(* LS Electric XG5000 project: 찐찐찐찐최종본_스마트홈_프로젝트_0225 *)
(* PLC LSPLC *)

(* Comments on direct variables
%MX0	램프0
%MX1	램프1
%MX2	램프2
%MX3	램프3
%MX4	색상조절변경버튼
%MX9	전원
%MX10	온도_자동
%MX11	 
%MX23	 
%MX29	따뜻한바람_1단계
%MX30	따뜻한바람_2단계
%MX31	따뜻한바람_3단계
%MX35	따뜻한바람_0단계
%MX172	 
%MX538	 
%MX709	전원
%MX710	온도_자동
%MX711	난방_수동_ON
%MX712	난방_수동_OFF
%MX713	난방_수동_RUN
%MX714	난방_자동_RUN
%MX715	난방기_ON
%MX721	냉방_수동_ON
%MX722	냉방_수동_OFF
%MX723	냉방_수동_RUN
%MX724	냉방_자동_RUN
%MX725	냉방기_ON
%MX726	난방기출력1
%MX727	냉방기출력1
%MX728	시간예약모드
%MX729	따뜻한바람_1단계
%MX730	따뜻한바람_2단계
%MX731	따뜻한바람_3단계
%MX732	시원한바람_1단계
%MX733	시원한바람_2단계
%MX734	시원한바람_3단계
%MX735	따뜻한바람_0단계
%MX736	시원한바람_0단계
%MX750	외출모드
%MX755	빈값
%MX760	보일러_전원
%MX761	보일러_자동_RUN
%MX762	보일러출력1
%MX763	보일러_온도조절_자동
%MX764	보일러_ON
%MX765	보일러_시간예약
%MX923	 
%MW10	조명색_변경
%MW100	셋팅온도
%MW101	온도_오차
%MW102	현재온도
%MW103	온도_오차1
%MW104	온도_오차2
%MW129	풍량
%MW200	밝기조절램프
%MW410	보일러_시간입력
%MW411	보일러_셋팅온도
%MW412	보일러_온도오차
%MW413	보일러_온도오차_덧셈
%MW414	보일러_온도오차_뺄셈
%MW415	현재온도
%MW416	보일러_표시데이터
%MW500	시간입력
%MW600	색상조절램프
*)

PROGRAM 조명 (* task: 스캔 프로그램 *)
VAR
    FF : FF;
    INST3 : R_TRIG;
    INST_사본1 : R_TRIG;
    INST_사본2 : R_TRIG;
    OFF AT %MX7 : BOOL;
    ON AT %MX8 : BOOL;
    밝기조절_1 AT %MX5 : BOOL;
    밝기조절_2 AT %MX6 : BOOL;
    시작 : BOOL;
    시작2 : BOOL;
    자기유지1 : BOOL;
    자기유지2 : BOOL;
    조명_1 AT %QX10 : BOOL;
    조명_2 AT %QX11 : BOOL;
    출력 : BOOL;
END_VAR
VAR
    _e1 : R_TRIG;
    _e2 : R_TRIG;
    _e3 : R_TRIG;
    _p4 : BOOL;
END_VAR

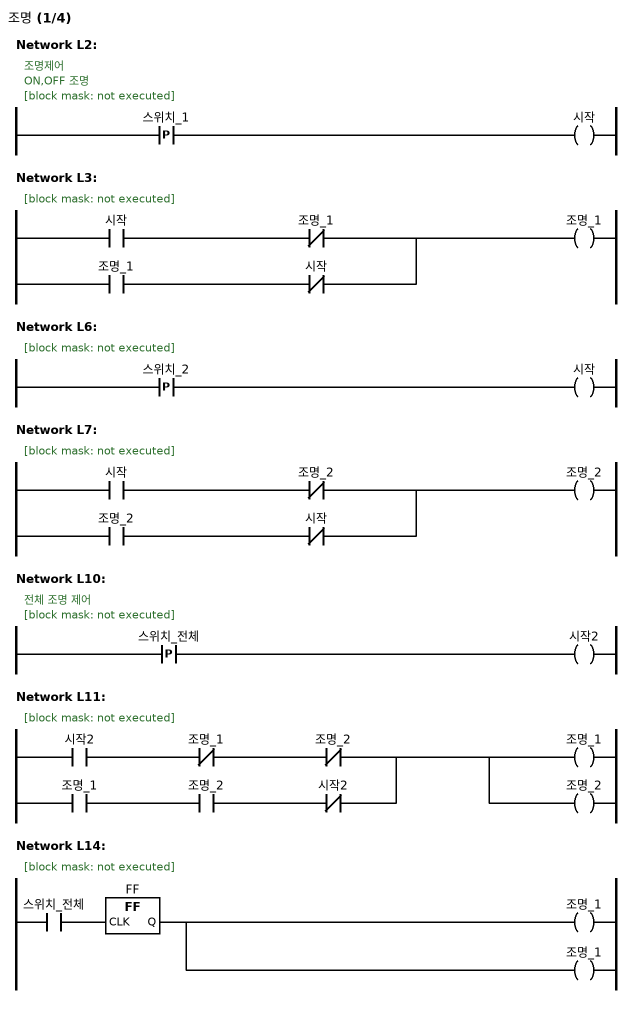
(* 조명제어 *)
(* ON,OFF 조명 *)
(* Rung L2 is block-masked: not executed *)
// _e1(CLK := 스위치_1);
// 시작 := _e1.Q;
(* Rung L3 is block-masked: not executed *)
// 조명_1 := (시작 AND NOT 조명_1) OR (조명_1 AND NOT 시작);
(* Rung L6 is block-masked: not executed *)
// _e2(CLK := 스위치_2);
// 시작 := _e2.Q;
(* Rung L7 is block-masked: not executed *)
// 조명_2 := (시작 AND NOT 조명_2) OR (조명_2 AND NOT 시작);
(* 전체 조명 제어 *)
(* Rung L10 is block-masked: not executed *)
// _e3(CLK := 스위치_전체);
// 시작2 := _e3.Q;
(* Rung L11 is block-masked: not executed *)
// _p4 := (시작2 AND NOT 조명_1 AND NOT 조명_2) OR (조명_1 AND 조명_2 AND NOT 시작2);
// 조명_1 := _p4;
// 조명_2 := _p4;
(* Rung L14 is block-masked: not executed *)
// FF(CLK := 스위치_전체);
// 조명_1 := FF.Q;
// 조명_1 := FF.Q;

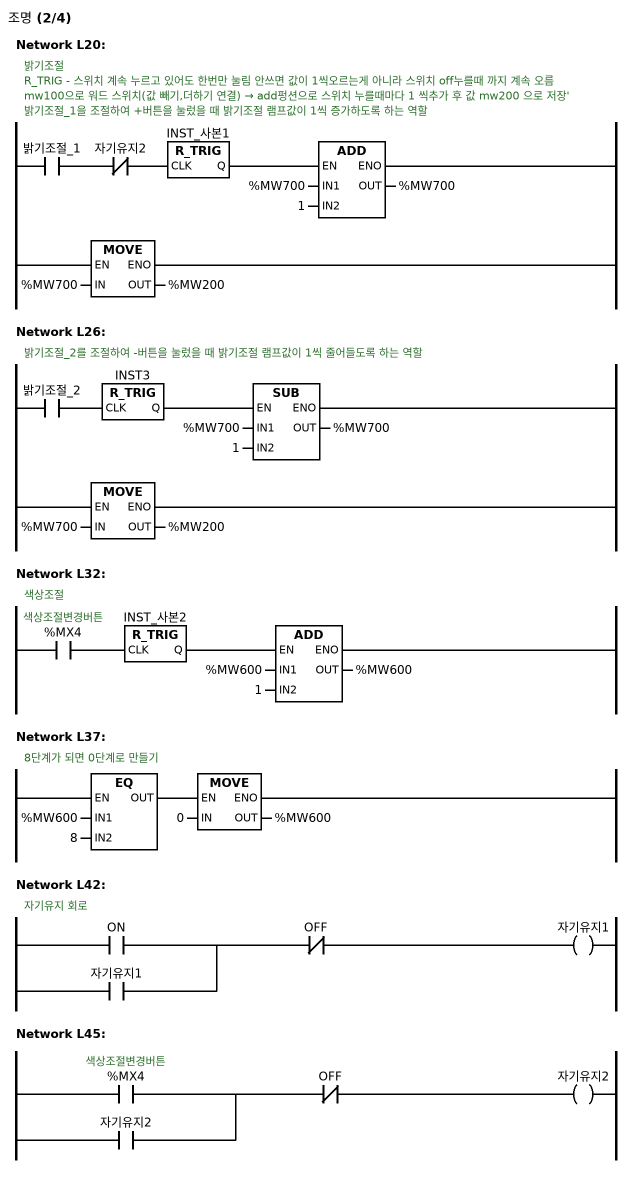
(* 밝기조절 *)
(* R_TRIG - 스위치 계속 누르고 있어도 한번만 눌림 안쓰면 값이 1씩오르는게 아니라 스위치 off누를때 까지 계속 오름 *)
(* mw100으로 워드 스위치(값 빼기,더하기 연결) → add펑션으로 스위치 누를때마다 1 씩추가 후 값 mw200 으로 저장' *)
(* 밝기조절_1을 조절하여 +버튼을 눌렀을 때 밝기조절 램프값이 1씩 증가하도록 하는 역할 *)
(* Rung L20 *)
INST_사본1(CLK := 밝기조절_1 AND NOT 자기유지2);
IF INST_사본1.Q THEN %MW700 := %MW700 + 1; END_IF;
%MW200 := %MW700;
(* 밝기조절_2를 조절하여 -버튼을 눌렀을 때 밝기조절 램프값이 1씩 줄어들도록 하는 역할 *)
(* Rung L26 *)
INST3(CLK := 밝기조절_2);
IF INST3.Q THEN %MW700 := %MW700 - 1; END_IF;
%MW200 := %MW700;
(* 색상조절 *)
(* Rung L32 *)
INST_사본2(CLK := %MX4);
IF INST_사본2.Q THEN %MW600 := %MW600 + 1; END_IF;
(* 8단계가 되면 0단계로 만들기 *)
(* Rung L37 *)
IF %MW600 = 8 THEN %MW600 := 0; END_IF;
(* 자기유지 회로 *)
(* Rung L42 *)
자기유지1 := (ON OR 자기유지1) AND NOT OFF;
(* Rung L45 *)
자기유지2 := (%MX4 OR 자기유지2) AND NOT OFF;

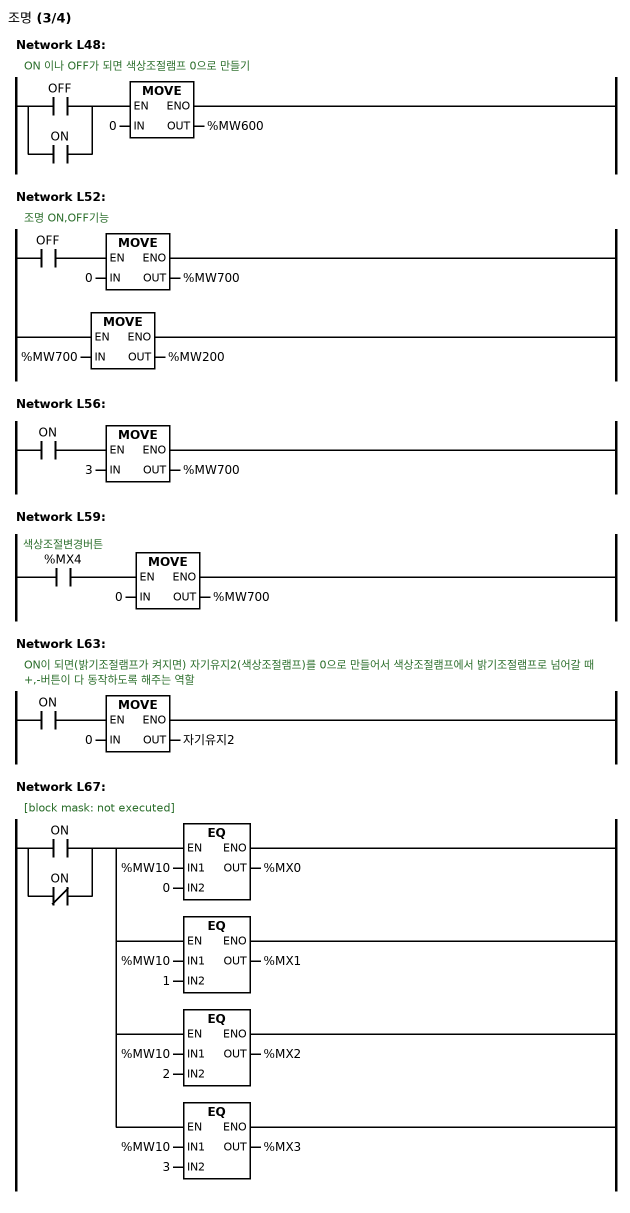
(* ON 이나 OFF가 되면 색상조절램프 0으로 만들기 *)
(* Rung L48 *)
IF OFF OR ON THEN %MW600 := 0; END_IF;
(* 조명 ON,OFF기능 *)
(* Rung L52 *)
IF OFF THEN %MW700 := 0; END_IF;
%MW200 := %MW700;
(* Rung L56 *)
IF ON THEN %MW700 := 3; END_IF;
(* Rung L59 *)
IF %MX4 THEN %MW700 := 0; END_IF;
(* ON이 되면(밝기조절램프가 켜지면) 자기유지2(색상조절램프)를 0으로 만들어서 색상조절램프에서 밝기조절램프로 넘어갈 때 +,-버튼이 다 동작하도록 해주는 역할 *)
(* Rung L63 *)
IF ON THEN 자기유지2 := 0; END_IF;
(* Rung L67 is block-masked: not executed *)
// IF ON OR NOT ON THEN
//     %MX0 := %MW10 = 0;
//     %MX1 := %MW10 = 1;
//     %MX2 := %MW10 = 2;
//     %MX3 := %MW10 = 3;
// END_IF;

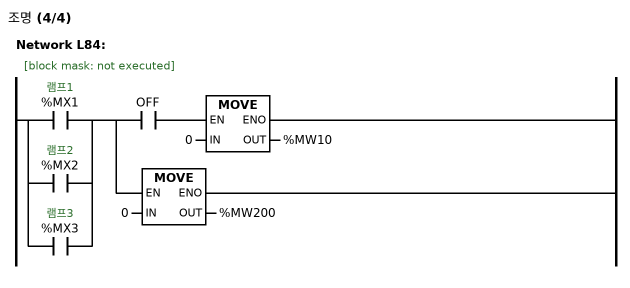
(* Rung L84 is block-masked: not executed *)
// IF (%MX1 OR %MX2 OR %MX3) AND OFF THEN %MW10 := 0; END_IF;
// IF %MX1 OR %MX2 OR %MX3 THEN %MW200 := 0; END_IF;
END_PROGRAM

PROGRAM 커튼 (* task: 스캔 프로그램 *)
VAR
    INST13 : TON;
    센서_커튼닫힘 AT %MX915 : BOOL;
    센서_커튼열림 AT %MX911 : BOOL;
    커튼_제어 AT %IX0.0.7 : BOOL;
    커튼_제어1 AT %IX0.0.8 : BOOL;
    커튼닫힘 AT %MX823 : BOOL;
    커튼열림 AT %MX822 : BOOL;
END_VAR
VAR
    _p1 : BOOL;
    _p2 : BOOL;
END_VAR

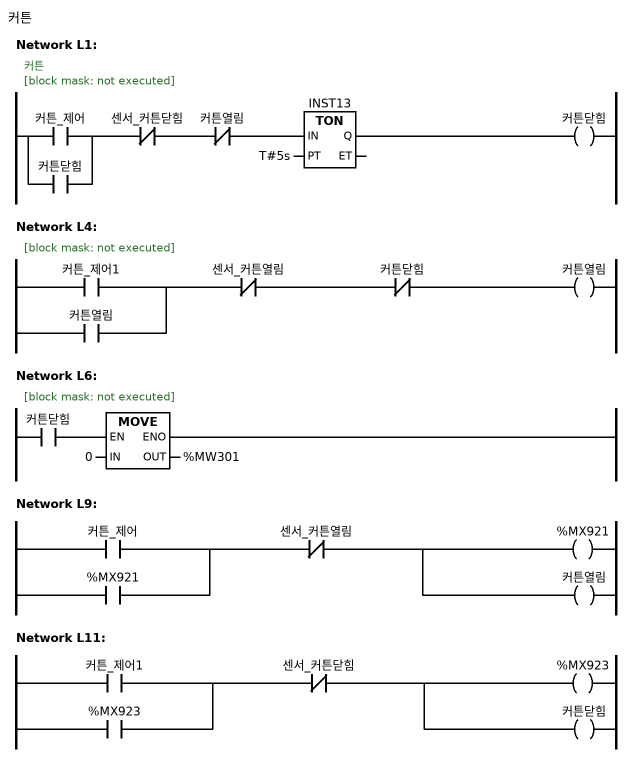
(* 커튼 *)
(* Rung L1 is block-masked: not executed *)
// INST13(IN := (커튼_제어 OR 커튼닫힘) AND NOT 센서_커튼닫힘 AND NOT 커튼열림, PT := T#5s);
// 커튼닫힘 := INST13.Q;
(* Rung L4 is block-masked: not executed *)
// 커튼열림 := (커튼_제어1 OR 커튼열림) AND NOT 센서_커튼열림 AND NOT 커튼닫힘;
(* Rung L6 is block-masked: not executed *)
// IF 커튼닫힘 THEN %MW301 := 0; END_IF;
(* Rung L9 *)
_p1 := (커튼_제어 OR %MX921) AND NOT 센서_커튼열림;
%MX921 := _p1;
커튼열림 := _p1;
(* Rung L11 *)
_p2 := (커튼_제어1 OR %MX923) AND NOT 센서_커튼닫힘;
%MX923 := _p2;
커튼닫힘 := _p2;
END_PROGRAM

PROGRAM 공동현관 (* task: 스캔 프로그램 *)
VAR
    INST10 : TON;
    INST12 : TON;
    INST9 : TON;
    공동현관_엘베 AT %MX8718 : BOOL;
    도어닫힘 AT %MX523 : BOOL;
    도어열림 AT %MX522 : BOOL;
    변환 : UDINT;
    센서_1층 AT %MX511 : BOOL;
    센서_도어열림 AT %MX516 : BOOL;
    센서_현관도어닫힘 AT %MX617 : BOOL;
    센서_현관도어열림 AT %MX616 : BOOL;
    현관도어닫힘 AT %MX623 : BOOL;
    현관도어열림 AT %MX622 : BOOL;
    호출_1층상승 AT %MX538 : BOOL;
END_VAR
VAR
    _p1 : BOOL;
    _t2 : BOOL;
    _t3 : BOOL;
    _t4 : BOOL;
    _t5 : BOOL;
END_VAR

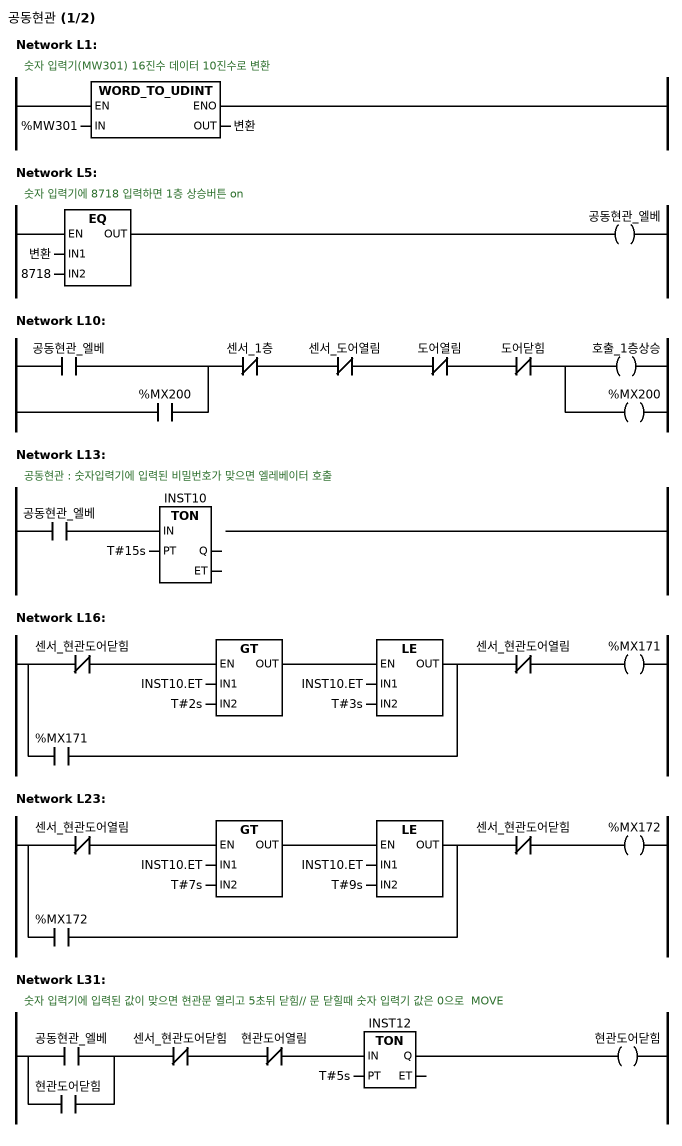
(* 숫자 입력기(MW301) 16진수 데이터 10진수로 변환 *)
(* Rung L1 *)
변환 := WORD_TO_UDINT(%MW301);
(* 숫자 입력기에 8718 입력하면 1층 상승버튼 on *)
(* Rung L5 *)
공동현관_엘베 := 변환 = 8718;
(* Rung L10 *)
_p1 := (공동현관_엘베 OR %MX200) AND NOT 센서_1층 AND NOT 센서_도어열림 AND NOT 도어열림 AND NOT 도어닫힘;
호출_1층상승 := _p1;
%MX200 := _p1;
(* 공동현관 : 숫자입력기에 입력된 비밀번호가 맞으면 엘레베이터 호출 *)
(* Rung L13 *)
INST10(IN := 공동현관_엘베, PT := T#15s);
(* Rung L16 *)
IF NOT 센서_현관도어닫힘 THEN _t2 := INST10.ET > T#2s; END_IF;
IF _t2 THEN _t3 := INST10.ET <= T#3s; END_IF;
%MX171 := (_t3 OR %MX171) AND NOT 센서_현관도어열림;
(* Rung L23 *)
IF NOT 센서_현관도어열림 THEN _t4 := INST10.ET > T#7s; END_IF;
IF _t4 THEN _t5 := INST10.ET <= T#9s; END_IF;
%MX172 := (_t5 OR %MX172) AND NOT 센서_현관도어닫힘;
(* 숫자 입력기에 입력된 값이 맞으면 현관문 열리고 5초뒤 닫힘// 문 닫힐때 숫자 입력기 값은 0으로  MOVE *)
(* Rung L31 *)
INST12(IN := (공동현관_엘베 OR 현관도어닫힘) AND NOT 센서_현관도어닫힘 AND NOT 현관도어열림, PT := T#5s);
현관도어닫힘 := INST12.Q;

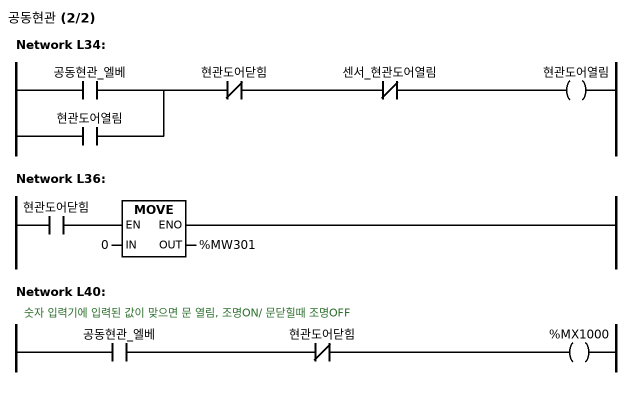
(* Rung L34 *)
현관도어열림 := (공동현관_엘베 OR 현관도어열림) AND NOT 현관도어닫힘 AND NOT 센서_현관도어열림;
(* Rung L36 *)
IF 현관도어닫힘 THEN %MW301 := 0; END_IF;
(* 숫자 입력기에 입력된 값이 맞으면 문 열림, 조명ON/ 문닫힐때 조명OFF *)
(* Rung L40 *)
%MX1000 := 공동현관_엘베 AND NOT 현관도어닫힘;
END_PROGRAM

PROGRAM 엘레베이터 (* task: 스캔 프로그램 *)
VAR
    INST : TON;
    INST1 : TON;
    INST9 : TON;
    공동현관_엘베 AT %MX8718 : BOOL;
    도어닫힘 AT %MX523 : BOOL;
    도어열림 AT %MX522 : BOOL;
    룸_1층 AT %MX501 : BOOL;
    룸_2층 AT %MX502 : BOOL;
    룸_3층 AT %MX503 : BOOL;
    룸_4층 AT %MX504 : BOOL;
    룸_5층 AT %MX505 : BOOL;
    룸_닫힘 AT %MX507 : BOOL;
    룸_비상 AT %MX500 : BOOL;
    룸_열림 AT %MX506 : BOOL;
    룸상승 AT %MX520 : BOOL;
    룸하강 AT %MX521 : BOOL;
    변환 : UDINT;
    상승램프 AT %MX524 : BOOL;
    센서_1층 AT %MX511 : BOOL;
    센서_2층 AT %MX512 : BOOL;
    센서_3층 AT %MX513 : BOOL;
    센서_4층 AT %MX514 : BOOL;
    센서_5층 AT %MX515 : BOOL;
    센서_도어닫힘 AT %MX517 : BOOL;
    센서_도어열림 AT %MX516 : BOOL;
    센서_현관도어닫힘 AT %MX617 : BOOL;
    센서_현관도어열림 AT %MX616 : BOOL;
    하강램프 AT %MX525 : BOOL;
    호출_1층상승 AT %MX538 : BOOL;
    호출_2층상승 AT %MX539 : BOOL;
    호출_2층하강 AT %MX542 : BOOL;
    호출_3층상승 AT %MX540 : BOOL;
    호출_3층하강 AT %MX543 : BOOL;
    호출_4층상승 AT %MX541 : BOOL;
    호출_4층하강 AT %MX544 : BOOL;
    호출_5층하강 AT %MX545 : BOOL;
END_VAR
VAR
    _e1 : R_TRIG;
    _e2 : R_TRIG;
    _e3 : R_TRIG;
    _e4 : R_TRIG;
    _e5 : R_TRIG;
    _t6 : BOOL;
    _t7 : BOOL;
    _t8 : BOOL;
    _t9 : BOOL;
    _p10 : BOOL;
    _p11 : BOOL;
END_VAR

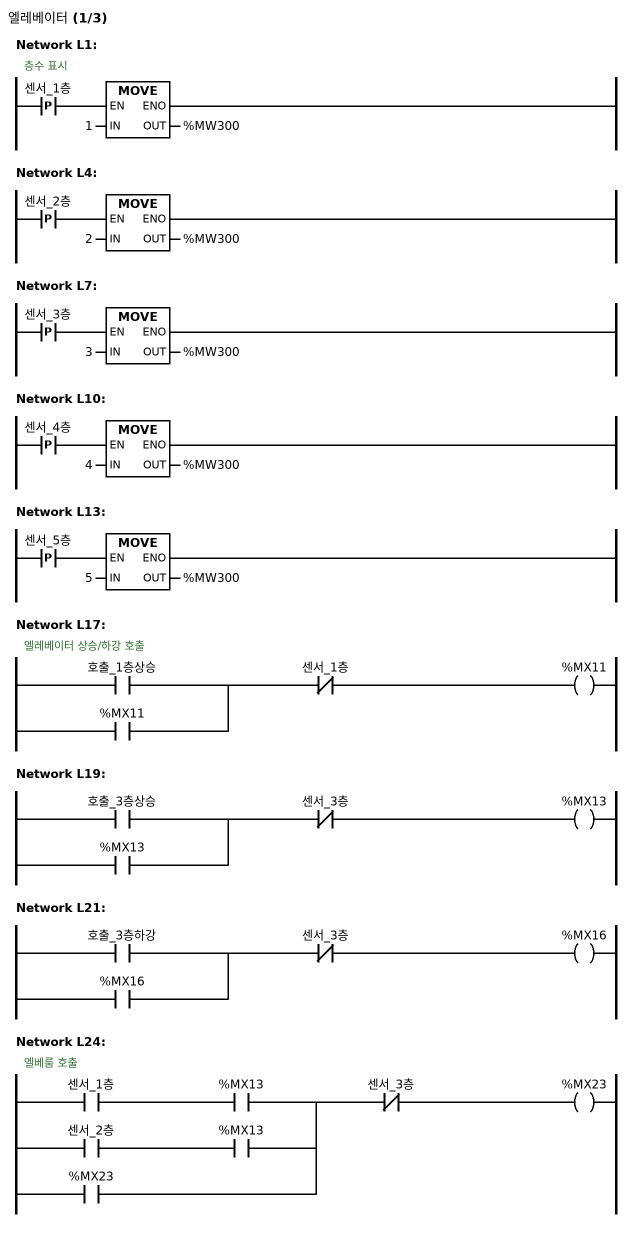
(* 층수 표시 *)
(* Rung L1 *)
_e1(CLK := 센서_1층);
IF _e1.Q THEN %MW300 := 1; END_IF;
(* Rung L4 *)
_e2(CLK := 센서_2층);
IF _e2.Q THEN %MW300 := 2; END_IF;
(* Rung L7 *)
_e3(CLK := 센서_3층);
IF _e3.Q THEN %MW300 := 3; END_IF;
(* Rung L10 *)
_e4(CLK := 센서_4층);
IF _e4.Q THEN %MW300 := 4; END_IF;
(* Rung L13 *)
_e5(CLK := 센서_5층);
IF _e5.Q THEN %MW300 := 5; END_IF;
(* 엘레베이터 상승/하강 호출 *)
(* Rung L17 *)
%MX11 := (호출_1층상승 OR %MX11) AND NOT 센서_1층;
(* Rung L19 *)
%MX13 := (호출_3층상승 OR %MX13) AND NOT 센서_3층;
(* Rung L21 *)
%MX16 := (호출_3층하강 OR %MX16) AND NOT 센서_3층;
(* 엘베룸 호출 *)
(* Rung L24 *)
%MX23 := ((센서_1층 AND %MX13) OR (센서_2층 AND %MX13) OR %MX23) AND NOT 센서_3층;

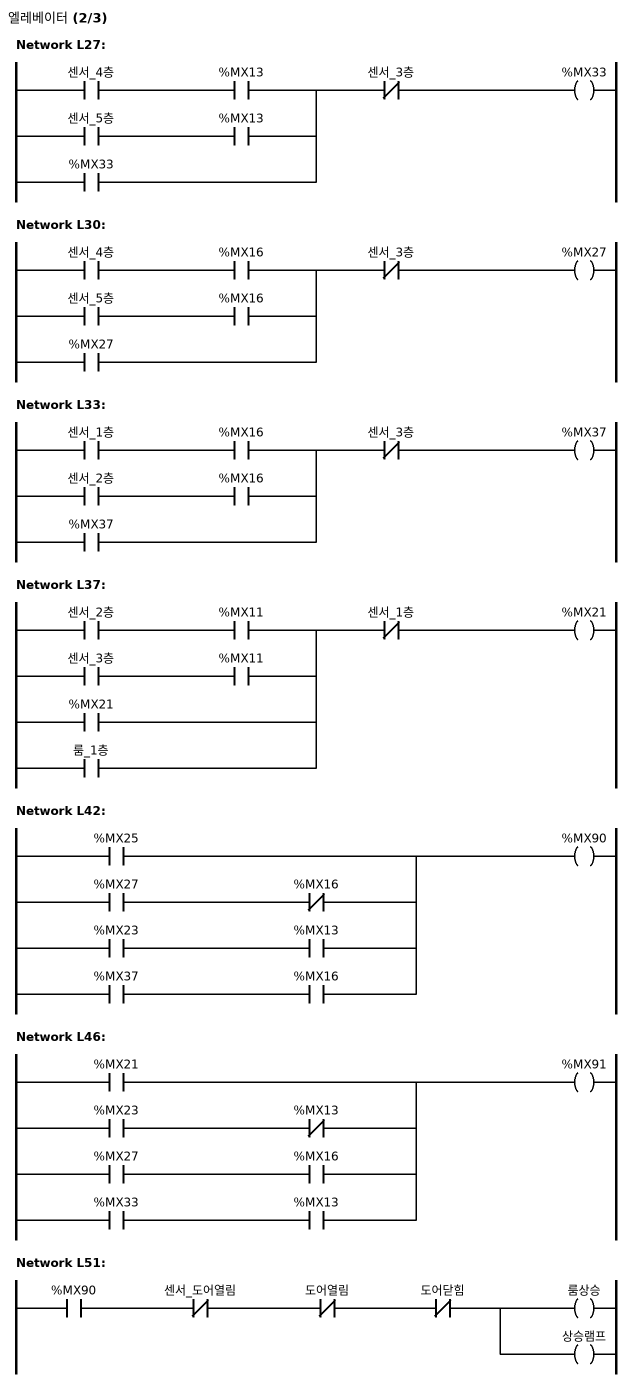
(* Rung L27 *)
%MX33 := ((센서_4층 AND %MX13) OR (센서_5층 AND %MX13) OR %MX33) AND NOT 센서_3층;
(* Rung L30 *)
%MX27 := ((센서_4층 AND %MX16) OR (센서_5층 AND %MX16) OR %MX27) AND NOT 센서_3층;
(* Rung L33 *)
%MX37 := ((센서_1층 AND %MX16) OR (센서_2층 AND %MX16) OR %MX37) AND NOT 센서_3층;
(* Rung L37 *)
%MX21 := ((센서_2층 AND %MX11) OR (센서_3층 AND %MX11) OR %MX21 OR 룸_1층) AND NOT 센서_1층;
(* Rung L42 *)
%MX90 := %MX25 OR (%MX27 AND NOT %MX16) OR (%MX23 AND %MX13) OR (%MX37 AND %MX16);
(* Rung L46 *)
%MX91 := %MX21 OR (%MX23 AND NOT %MX13) OR (%MX27 AND %MX16) OR (%MX33 AND %MX13);
(* Rung L51 *)
룸상승 := %MX90 AND NOT 센서_도어열림 AND NOT 도어열림 AND NOT 도어닫힘;
상승램프 := %MX90 AND NOT 센서_도어열림 AND NOT 도어열림 AND NOT 도어닫힘;

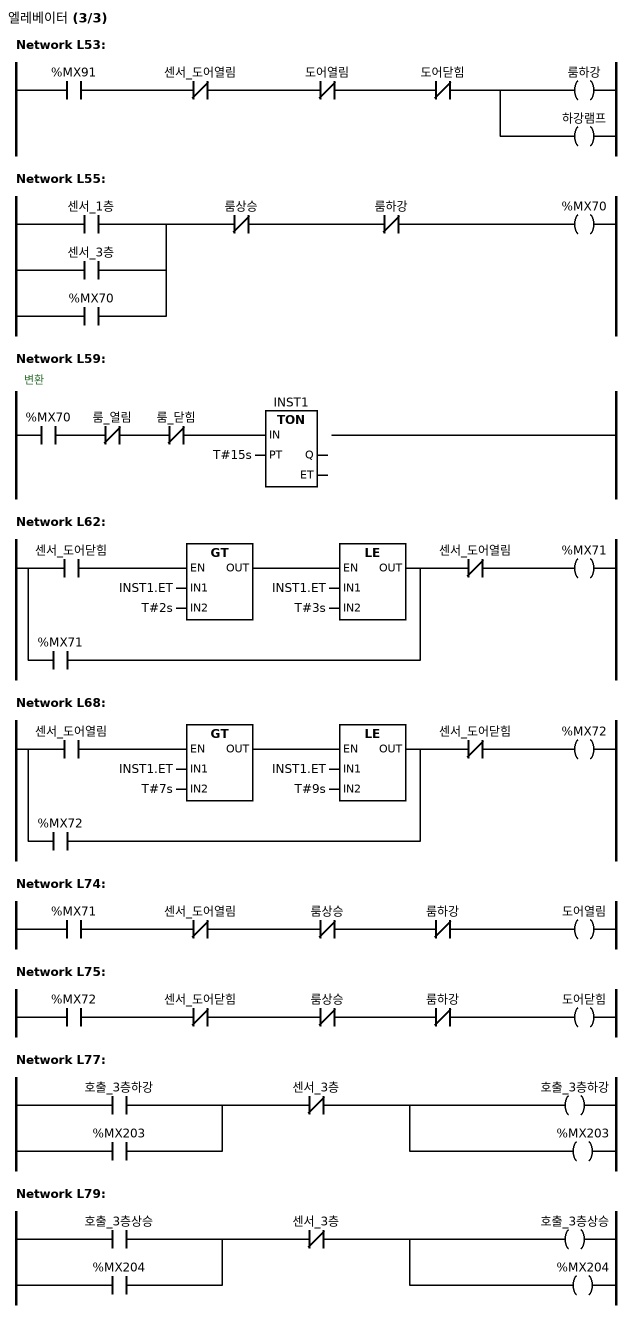
(* Rung L53 *)
룸하강 := %MX91 AND NOT 센서_도어열림 AND NOT 도어열림 AND NOT 도어닫힘;
하강램프 := %MX91 AND NOT 센서_도어열림 AND NOT 도어열림 AND NOT 도어닫힘;
(* Rung L55 *)
%MX70 := (센서_1층 OR 센서_3층 OR %MX70) AND NOT 룸상승 AND NOT 룸하강;
(* 변환 *)
(* Rung L59 *)
INST1(IN := %MX70 AND NOT 룸_열림 AND NOT 룸_닫힘, PT := T#15s);
(* Rung L62 *)
IF 센서_도어닫힘 THEN _t6 := INST1.ET > T#2s; END_IF;
IF _t6 THEN _t7 := INST1.ET <= T#3s; END_IF;
%MX71 := (_t7 OR %MX71) AND NOT 센서_도어열림;
(* Rung L68 *)
IF 센서_도어열림 THEN _t8 := INST1.ET > T#7s; END_IF;
IF _t8 THEN _t9 := INST1.ET <= T#9s; END_IF;
%MX72 := (_t9 OR %MX72) AND NOT 센서_도어닫힘;
(* Rung L74 *)
도어열림 := %MX71 AND NOT 센서_도어열림 AND NOT 룸상승 AND NOT 룸하강;
(* Rung L75 *)
도어닫힘 := %MX72 AND NOT 센서_도어닫힘 AND NOT 룸상승 AND NOT 룸하강;
(* Rung L77 *)
_p10 := (호출_3층하강 OR %MX203) AND NOT 센서_3층;
호출_3층하강 := _p10;
%MX203 := _p10;
(* Rung L79 *)
_p11 := (호출_3층상승 OR %MX204) AND NOT 센서_3층;
호출_3층상승 := _p11;
%MX204 := _p11;
END_PROGRAM

PROGRAM 가스제어 (* task: 스캔 프로그램 *)
VAR
    div_값 : UDINT;
    E0 AT %IX0.0.0 : BOOL; (* 전기 입력 *)
    int변경 : UDINT;
    LED상태 AT %QX0.1.1 : BOOL;
    LED유지 AT %MX0 : BOOL;
    LNG가스누출 : BOOL;
    Timer : TON;
    time변경 : UDINT;
    udint변경 : UDINT;
    가스 AT %QX0.1.2 : BOOL;
    가스레인지 AT %QX0.1.3 : BOOL;
    가스레인지버튼 AT %IX0.0.3 : BOOL;
    가스밸브 AT %IX0.0.2 : BOOL;
    가스센서 : BOOL;
    가스유지 AT %MX1 : BOOL;
    누출감지 AT %QX0.1.4 : BOOL;
    누출감지시작 : BOOL;
    두꺼비집 AT %IX0.0.1 : BOOL;
    메모리값 : INT;
    밀리변경 : INT;
    시간 : TIME;
    전기ON AT %QX0.1.0 : BOOL;
    카운터 : TIME;
END_VAR
VAR
    _e1 : R_TRIG;
    _p2 : BOOL;
END_VAR

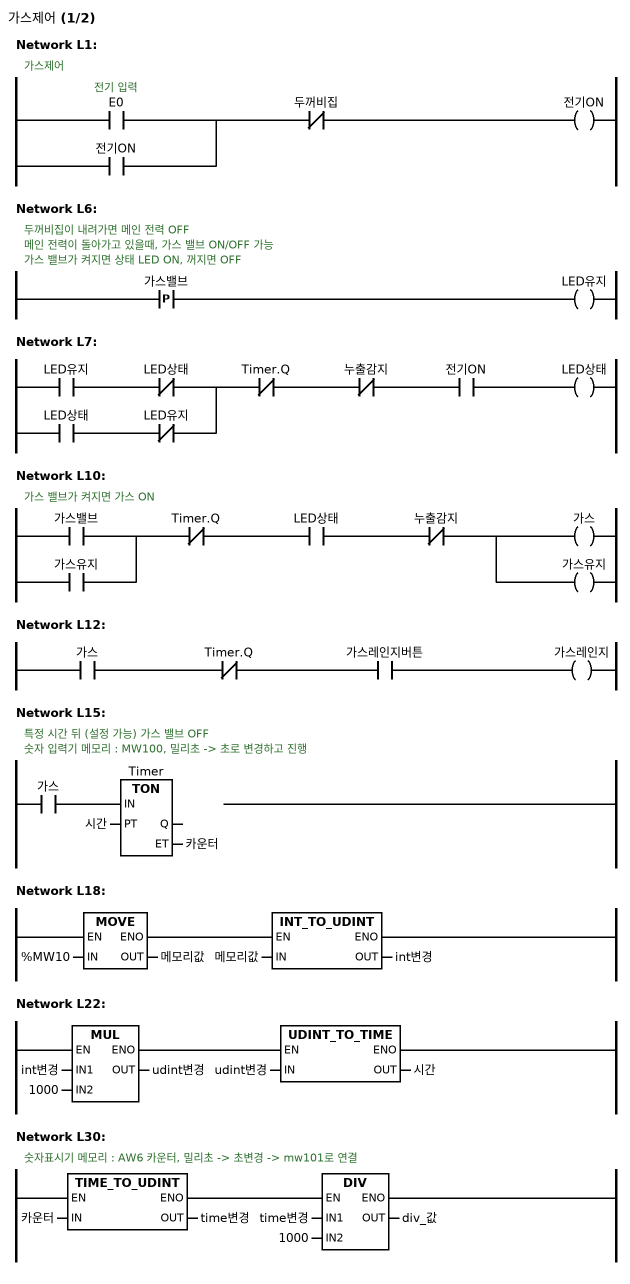
(* 가스제어 *)
(* Rung L1 *)
전기ON := (E0 OR 전기ON) AND NOT 두꺼비집;
(* 두꺼비집이 내려가면 메인 전력 OFF *)
(* 메인 전력이 돌아가고 있을때, 가스 밸브 ON/OFF 가능 *)
(* 가스 밸브가 켜지면 상태 LED ON, 꺼지면 OFF *)
(* Rung L6 *)
_e1(CLK := 가스밸브);
LED유지 := _e1.Q;
(* Rung L7 *)
LED상태 := ((LED유지 AND NOT LED상태) OR (LED상태 AND NOT LED유지)) AND NOT Timer.Q AND NOT 누출감지 AND 전기ON;
(* 가스 밸브가 켜지면 가스 ON *)
(* Rung L10 *)
_p2 := (가스밸브 OR 가스유지) AND NOT Timer.Q AND LED상태 AND NOT 누출감지;
가스 := _p2;
가스유지 := _p2;
(* Rung L12 *)
가스레인지 := 가스 AND NOT Timer.Q AND 가스레인지버튼;
(* 특정 시간 뒤 (설정 가능) 가스 밸브 OFF *)
(* 숫자 입력기 메모리 : MW100, 밀리초 -> 초로 변경하고 진행 *)
(* Rung L15 *)
Timer(IN := 가스, PT := 시간, ET => 카운터);
(* Rung L18 *)
메모리값 := %MW10;
int변경 := INT_TO_UDINT(메모리값);
(* Rung L22 *)
udint변경 := int변경 * 1000;
시간 := UDINT_TO_TIME(udint변경);
(* 숫자표시기 메모리 : AW6 카운터, 밀리초 -> 초변경 -> mw101로 연결 *)
(* Rung L30 *)
time변경 := TIME_TO_UDINT(카운터);
div_값 := time변경 / 1000;

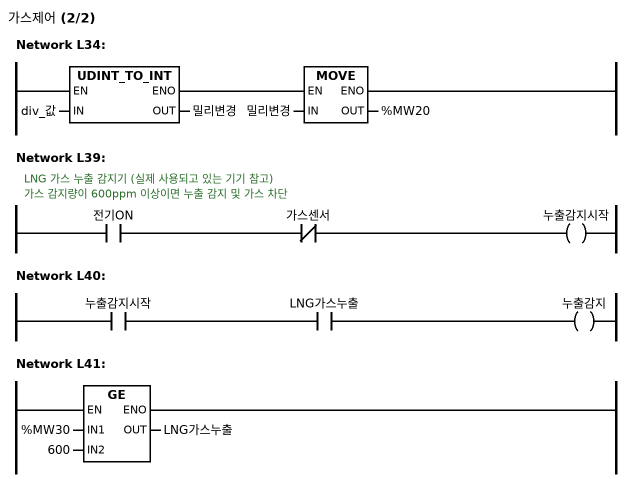
(* Rung L34 *)
밀리변경 := UDINT_TO_INT(div_값);
%MW20 := 밀리변경;
(* LNG 가스 누출 감지기 (실제 사용되고 있는 기기 참고) *)
(* 가스 감지량이 600ppm 이상이면 누출 감지 및 가스 차단 *)
(* Rung L39 *)
누출감지시작 := 전기ON AND NOT 가스센서;
(* Rung L40 *)
누출감지 := 누출감지시작 AND LNG가스누출;
(* Rung L41 *)
LNG가스누출 := %MW30 >= 600;
END_PROGRAM

PROGRAM 보일러 (* task: 스캔 프로그램 *)
VAR
    시간입력변환2 : TIME;
    출력_2 : UDINT;
    타이머4 : TON;
END_VAR

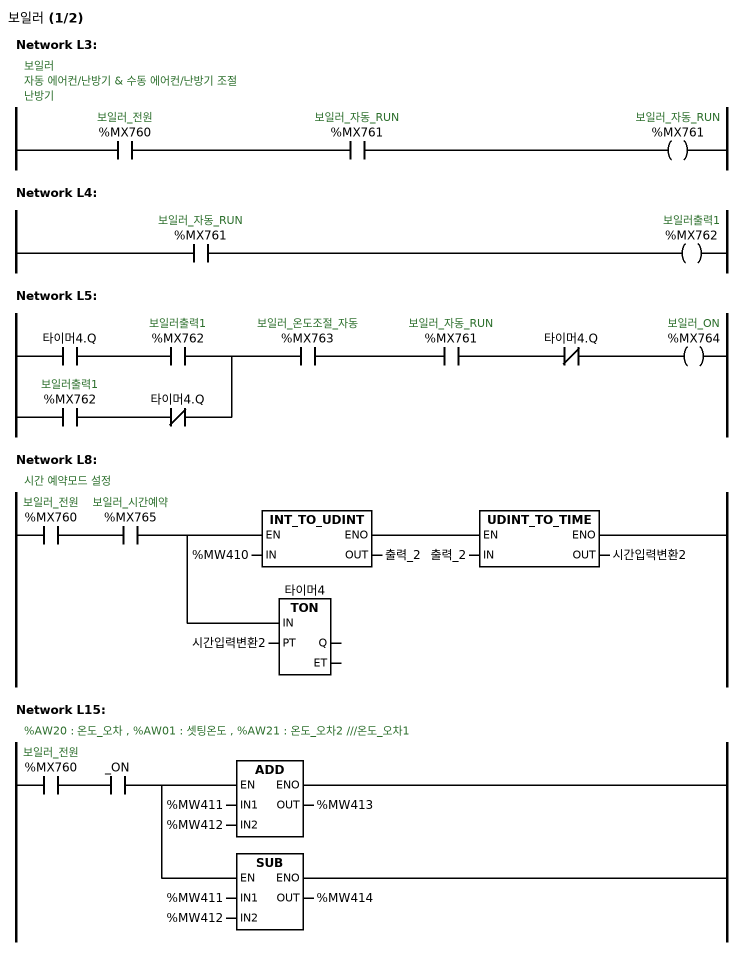
(* 보일러 *)
(* 자동 에어컨/난방기 & 수동 에어컨/난방기 조절 *)
(* 난방기 *)
(* Rung L3 *)
%MX761 := %MX760 AND %MX761;
(* Rung L4 *)
%MX762 := %MX761;
(* Rung L5 *)
%MX764 := ((타이머4.Q AND %MX762) OR (%MX762 AND NOT 타이머4.Q)) AND %MX763 AND %MX761 AND NOT 타이머4.Q;
(* 시간 예약모드 설정 *)
(* Rung L8 *)
IF %MX760 AND %MX765 THEN
    출력_2 := INT_TO_UDINT(%MW410);
    시간입력변환2 := UDINT_TO_TIME(출력_2);
END_IF;
타이머4(IN := %MX760 AND %MX765, PT := 시간입력변환2);
(* %AW20 : 온도_오차 , %AW01 : 셋팅온도 , %AW21 : 온도_오차2 ///온도_오차1 *)
(* Rung L15 *)
IF %MX760 AND _ON THEN
    %MW413 := %MW411 + %MW412;
    %MW414 := %MW411 - %MW412;
END_IF;

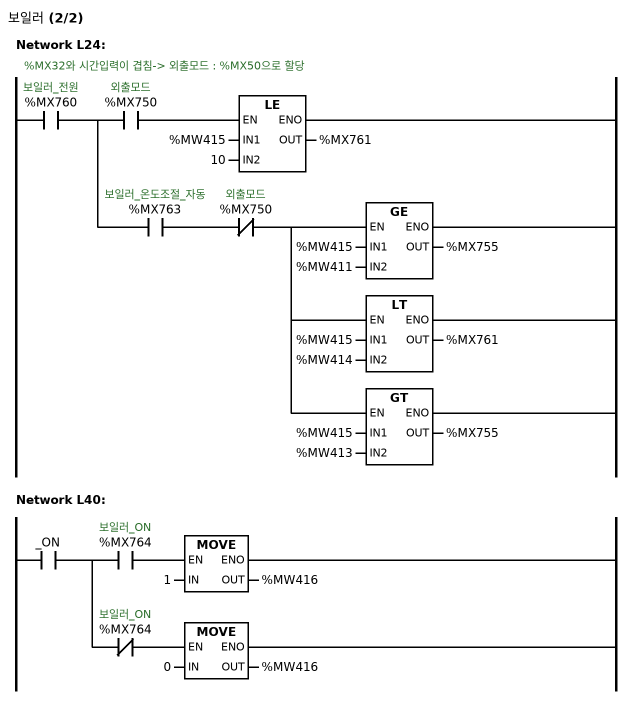
(* %MX32와 시간입력이 겹침-> 외출모드 : %MX50으로 할당 *)
(* Rung L24 *)
IF %MX760 AND %MX750 THEN %MX761 := %MW415 <= 10; END_IF;
IF %MX760 AND %MX763 AND NOT %MX750 THEN
    %MX755 := %MW415 >= %MW411;
    %MX761 := %MW415 < %MW414;
    %MX755 := %MW415 > %MW413;
END_IF;
(* Rung L40 *)
IF _ON AND %MX764 THEN %MW416 := 1; END_IF;
IF _ON AND NOT %MX764 THEN %MW416 := 0; END_IF;
END_PROGRAM

PROGRAM 냉난방기 (* task: 스캔 프로그램 *)
VAR
    시간입력변환 : TIME;
    출력_1 : UDINT;
    타이머3 : TON;
END_VAR
VAR
    _e1 : R_TRIG;
    _e2 : R_TRIG;
    _p3 : BOOL;
    _p4 : BOOL;
END_VAR

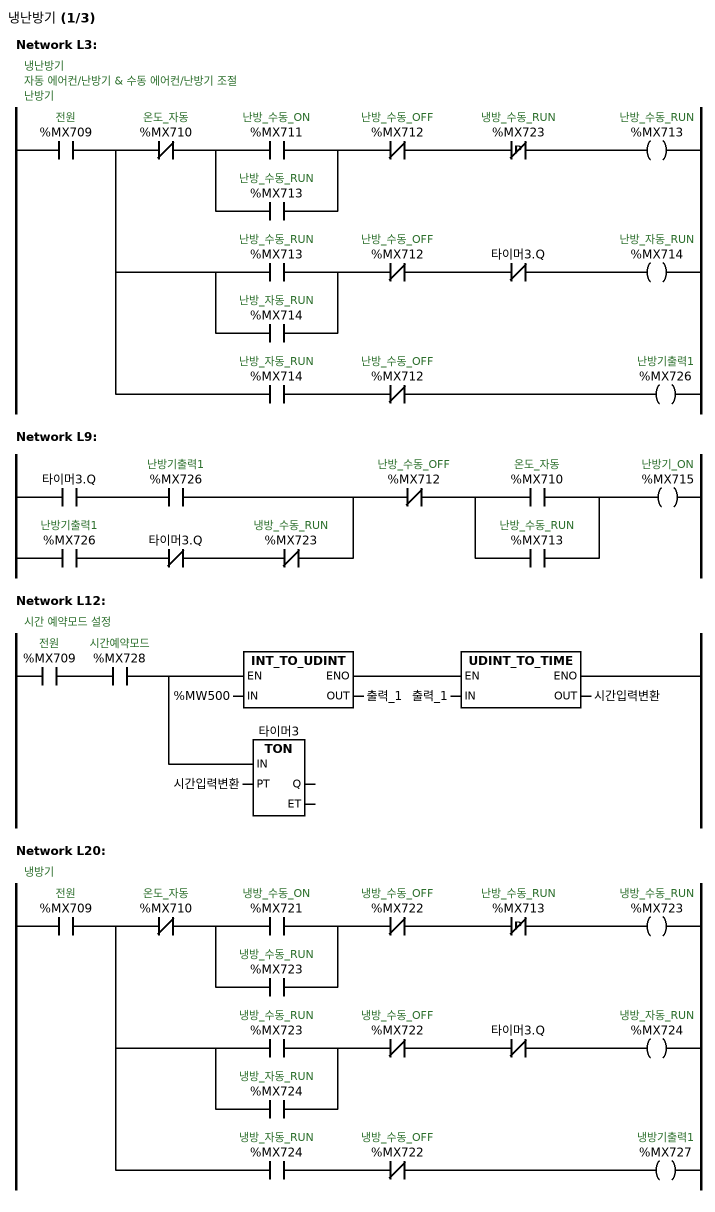
(* 냉난방기 *)
(* 자동 에어컨/난방기 & 수동 에어컨/난방기 조절 *)
(* 난방기 *)
(* Rung L3 *)
_e1(CLK := %MX723);
%MX713 := %MX709 AND NOT %MX710 AND (%MX711 OR %MX713) AND NOT %MX712 AND NOT _e1.Q;
%MX714 := %MX709 AND (%MX713 OR %MX714) AND NOT %MX712 AND NOT 타이머3.Q;
%MX726 := %MX709 AND %MX714 AND NOT %MX712;
(* Rung L9 *)
%MX715 := ((타이머3.Q AND %MX726) OR (%MX726 AND NOT 타이머3.Q AND NOT %MX723)) AND NOT %MX712 AND (%MX710 OR %MX713);
(* 시간 예약모드 설정 *)
(* Rung L12 *)
IF %MX709 AND %MX728 THEN
    출력_1 := INT_TO_UDINT(%MW500);
    시간입력변환 := UDINT_TO_TIME(출력_1);
END_IF;
타이머3(IN := %MX709 AND %MX728, PT := 시간입력변환);
(* 냉방기 *)
(* Rung L20 *)
_e2(CLK := %MX713);
%MX723 := %MX709 AND NOT %MX710 AND (%MX721 OR %MX723) AND NOT %MX722 AND NOT _e2.Q;
%MX724 := %MX709 AND (%MX723 OR %MX724) AND NOT %MX722 AND NOT 타이머3.Q;
%MX727 := %MX709 AND %MX724 AND NOT %MX722;

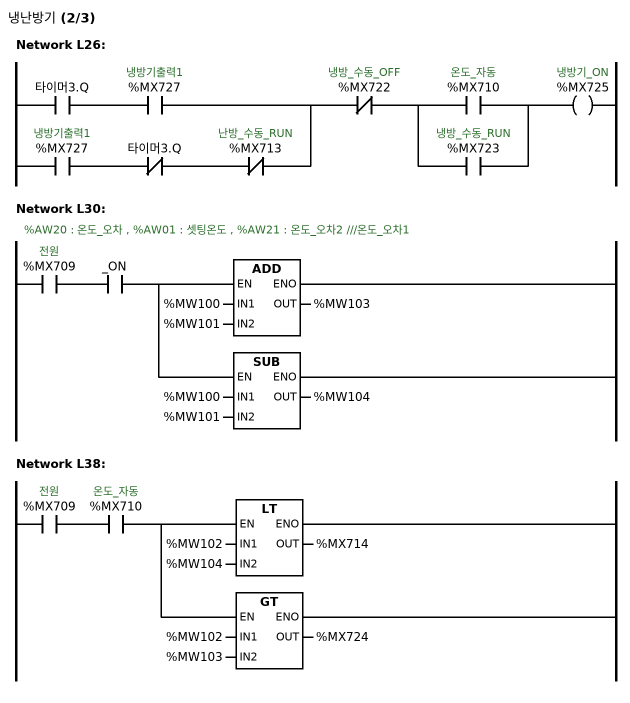
(* Rung L26 *)
%MX725 := ((타이머3.Q AND %MX727) OR (%MX727 AND NOT 타이머3.Q AND NOT %MX713)) AND NOT %MX722 AND (%MX710 OR %MX723);
(* %AW20 : 온도_오차 , %AW01 : 셋팅온도 , %AW21 : 온도_오차2 ///온도_오차1 *)
(* Rung L30 *)
IF %MX709 AND _ON THEN
    %MW103 := %MW100 + %MW101;
    %MW104 := %MW100 - %MW101;
END_IF;
(* Rung L38 *)
IF %MX709 AND %MX710 THEN
    %MX714 := %MW102 < %MW104;
    %MX724 := %MW102 > %MW103;
END_IF;

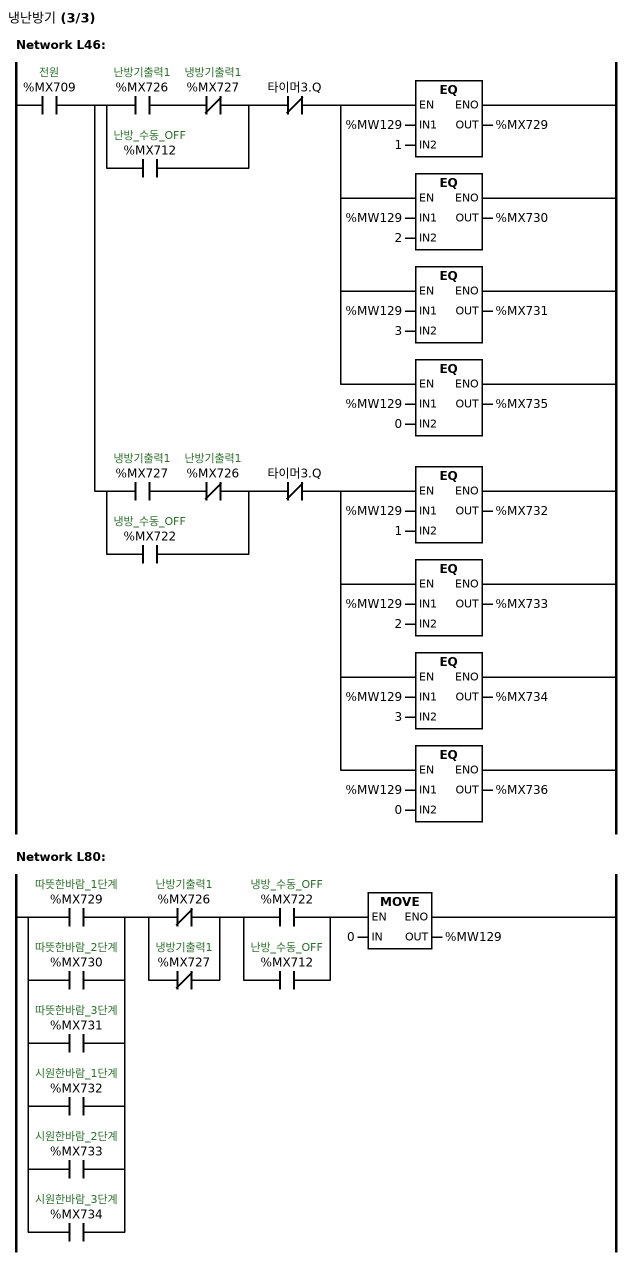
(* Rung L46 *)
_p3 := %MX709 AND ((%MX726 AND NOT %MX727) OR %MX712) AND NOT 타이머3.Q;
IF _p3 THEN
    %MX729 := %MW129 = 1;
    %MX730 := %MW129 = 2;
    %MX731 := %MW129 = 3;
    %MX735 := %MW129 = 0;
END_IF;
_p4 := %MX709 AND ((%MX727 AND NOT %MX726) OR %MX722) AND NOT 타이머3.Q;
IF _p4 THEN
    %MX732 := %MW129 = 1;
    %MX733 := %MW129 = 2;
    %MX734 := %MW129 = 3;
    %MX736 := %MW129 = 0;
END_IF;
(* Rung L80 *)
IF (%MX729 OR %MX730 OR %MX731 OR %MX732 OR %MX733 OR %MX734) AND (NOT %MX726 OR NOT %MX727) AND (%MX722 OR %MX712) THEN
    %MW129 := 0;
END_IF;
END_PROGRAM